INTERFACE EncodedDrive

METHOD moveAbsolute : BOOL
VAR_INPUT
	newTarget : LREAL; 
END_VAR
END_METHOD

METHOD moveRelative : BOOL
VAR_INPUT
	distance : LREAL;
END_VAR
END_METHOD

PROPERTY Position : LREAL
GET
END_GET
SET
END_SET
END_PROPERTY

PROPERTY TargetPosition : LREAL
GET
END_GET
SET
END_SET
END_PROPERTY

END_INTERFACE

(* stored: Version 1.1.0.1, ProductVersion 3.1.4024.11
   Itf EncodedDrive: Id {542dde8d-3f0e-453c-8c39-9501a69f7da7}
   Method moveAbsolute: Id {2c02535f-adbe-4dfa-ac4b-ddfb412f57da}
   Method moveRelative: Id {83781e94-128b-41f5-8391-03ac83176760}
   Property Position: Id {5fd6800f-0c34-471b-a53d-c6651be10b18}
   Get Get: Id {909a548f-7b4d-4e90-9a92-b28803717256}
   Set Set: Id {c69dd791-2b1e-43cf-bdbc-401b895c70cd}
   Property TargetPosition: Id {271e05ba-4585-4f4a-bb6c-097f79560249}
   Get Get: Id {bf4acaac-8701-405d-be0c-eaf98075daeb}
   Set Set: Id {41973d7f-5019-4ad3-ab11-fe1316916a7d} *)
